TYPE ST_Torque :
STRUCT
	Invert:LREAL;
	PosReq:UINT;
	NegReq:UINT;
END_STRUCT
END_TYPE

(* stored: Version 1.1.0.1, ProductVersion 3.1.4024.11
   DUT ST_Torque: Id {a97e683c-584d-4de5-ab84-586fdcdac054} *)
